// TIA Portal V20 export
TYPE "UDT_MTP_StringProcessValueIn"
   STRUCT
      WQC { ExternalWritable := 'False'} : Byte := 16#FF;   // Worst Quality Code
      V : String[40];   // Value
      VQC : Byte := 16#FF;   // Quality Code of the current received value
   END_STRUCT;
END_TYPE
